(* PLC project CodesysTest_empty.project, CODESYS CODESYS V3.5 SP17 Patch 3 *)
(* stored: creationDateTime 2022-04-24T22:05:35.9296647, modificationDateTime 2022-04-23T22:33:03.5422534 *)

PROGRAM POU

            
          
END_PROGRAM
